Staubli VAL3: Control_Loffset.pgx

public program Control_Loffset(num& x_nFrom, num& x_nTo)
  local string l_sItem[2]
  local num l_nNum
  local num l_nKey
  local num l_nData[6]
  local num l_nSelectIndex
begin

  //修改点位的 joint
l_nData[0]=x_nFrom
l_nData[1]=x_nTo

  l_sItem[0]="开始    :"+toString("",l_nData[0])
  l_sItem[1]="停止    :"+toString("",l_nData[1])
  call Control_BottomS(",,,,,,取消,确定")
  call Control_PanelXY(8,0,15,6)
  call Control_Panel("局部偏差值")
  call Control_List(l_sItem,l_nSelectIndex)
  while true
    l_nKey=getKey()

    switch l_nKey
      case 261
        l_nSelectIndex=max(0,l_nSelectIndex-1)
      break

      case 266
        l_nSelectIndex=min(l_nSelectIndex+1,1)
      break

      case 278
          x_nFrom=l_nData[0]
          x_nTo=l_nData[1]
         cls()
        return
      break


      case 277,255

        cls()
        return
      break

      case 270
        call Float_Edit(l_nData[l_nSelectIndex],nPanelLTopX+7,l_nSelectIndex+nPanelLTopY+1)
      break

    endSwitch

    if l_nKey!=-1
  l_sItem[0]="开始    :"+toString("",l_nData[0])
  l_sItem[1]="停止    :"+toString("",l_nData[1])
      call Control_List(l_sItem,l_nSelectIndex)

    endIf






  endWhile





end
